// TwinCAT 3 PLC project PLC1
// ProgramVersion: 3.1.4023.0
// libraries:
//   Tc2_Standard, * (Beckhoff Automation GmbH)
//   Tc2_System, * (Beckhoff Automation GmbH)
//   Tc2_Utilities, * (Beckhoff Automation GmbH)
//   Tc3_Database, * (Beckhoff Automation GmbH)
//   Tc3_EventLogger, * (Beckhoff Automation GmbH)
//   Tc3_Module, * (Beckhoff Automation GmbH)
// project tree:
//   / PlcTask.TcTTO
//   POUs/ MAIN.TcPOU
// real-time tasks:
//   TASK PlcTask: cycle T#10ms, priority 20, ADS port 350

CONFIGURATION PLC1
    RESOURCE PLC ON TwinCAT3
        TASK PlcTask(INTERVAL := T#10ms, PRIORITY := 20);
        PROGRAM MAIN WITH PlcTask : MAIN;
    END_RESOURCE
END_CONFIGURATION

// ---- POUs/MAIN.TcPOU
PROGRAM MAIN
VAR
	i: BYTE := 0;
	bStart: BOOL := TRUE;
	bLog: BOOL := FALSE;

	//Query Builder for Document DB
	fbNoSqlQueryBuilder_DocumentDB: FB_NoSQLQueryBuilder_DocumentDB;
	InsertQueryOption: T_QueryOptionDocumentDB_Insert;
	sDocument: STRING (1000);

	//Query Execution
	fbNoSqlQuery: FB_NoSQLQueryEvt(sNetID:= '', tTimeout:= T#5S);
	myDBID: UDINT := 1;
	TcMessage: I_TcMessage;
END_VAR

IF bStart THEN
	CreateQuery();
	bStart:= FALSE;
END_IF

IF bLog THEN
	CreateDocument();
	IF fbNoSqlQuery.Execute(hDBID:= myDBID, iNoSQLQueryBuilder:= fbNoSqlQueryBuilder_DocumentDB) THEN
		IF fbNoSqlQuery.bError THEN
			TcMessage:= fbNoSqlQuery.ipTcResult;
		END_IF
		bLog:= FALSE;
		i := i + 1;
	END_IF
END_IF

ACTION CreateDocument:
sDocument:= '{"name": "son",
				"position": "intern",
				"dateOfBirth": "27-07-1999",
				"number":';
sDocument := CONCAT(STR1:= sDocument, STR2:= BYTE_TO_STRING(i));
sDocument := CONCAT(STR1:= sDocument, STR2:= '}');
END_ACTION

ACTION CreateQuery:
InsertQueryOption.pDocuments := ADR(sDocument);
InsertQueryOption.cbDocuments := SIZEOF(sDocument);

fbNoSqlQueryBuilder_DocumentDB.eQueryType := E_DocumentDbQueryType.InsertOne;
fbNoSqlQueryBuilder_DocumentDB.sCollectionName := 'Customer';
fbNoSqlQueryBuilder_DocumentDB.pQueryOptions := ADR(InsertQueryOption);
fbNoSqlQueryBuilder_DocumentDB.cbQueryOptions := SIZEOF(InsertQueryOption);
END_ACTION

END_PROGRAM
